// TIA Portal project "scl_6" (V18)

(* hardware
DEVICE "S7-1200 station_1"  S7-1200 Station
   slot 0: "Rack_0"  S7-1200 Rack  Rack  V1.0
   slot 1: "PLC_1"  CPU 1214C DC/DC/DC  6ES7 214-1AG40-0XB0  V4.6
*)

// ===== PLC "PLC_1"  CPU 1214C DC/DC/DC =====

VAR_GLOBAL   // PLC tag table "Default tag table"
   "START" AT %I0.0 : Bool;
   "STOP" AT %I0.1 : Bool;
   "MOTOR" AT %Q0.0 : Bool;
   "START1" AT %I0.2 : Bool;
   "START2" AT %I0.3 : Bool;
   "START3" AT %I0.4 : Bool;
   "SICAKLIK" AT %IW64 : Word;
   "BASINÇ" AT %IW66 : Word;
   "VALF1" AT %Q0.1 : Bool;
   "VALF2" AT %Q0.2 : Bool;
   "VALF3" AT %Q0.3 : Bool;
   "VALF4" AT %Q0.4 : Bool;
   "VALF5" AT %Q0.5 : Bool;
   "VALF6" AT %Q0.6 : Bool;
   "VALF7" AT %Q0.7 : Bool;
END_VAR

VAR_GLOBAL   // PLC tag table "Tag table_1"
   "ANALOG DEĞER" AT %IW68 : Int;
   "ANALOG DEĞER(1)" AT %IW70 : Int;
   "VALF 1" AT %Q1.0 : Bool;
   "VALF 2" AT %Q1.1 : Bool;
   "VALF 3" AT %Q1.2 : Bool;
   "VALF 4" AT %Q1.3 : Bool;
   "VALF 5" AT %Q1.4 : Bool;
   "VALF 6" AT %Q1.5 : Bool;
   "VALF 7" AT %Q1.6 : Bool;
   "DİGİTAL ÇIKIŞLAR" AT %QW0 : Word;
END_VAR

FUNCTION "Block_1" : Void   // FC1, SCL
{ S7_Optimized_Access := 'TRUE' }
VERSION : 0.1
BEGIN
   IF "START"=1 THEN
       // Statement section IF
       "MOTOR" := 1;
   ELSE
       // Statement section ELSE
       "MOTOR" := 0;
   END_IF;
END_FUNCTION

FUNCTION "Block_2" : Void   // FC2, SCL
{ S7_Optimized_Access := 'TRUE' }
VERSION : 0.1
BEGIN
   IF "START1"=1 THEN
       "VALF1":=1;
   ELSIF "START2"=1 THEN
       "VALF2":=1;
   ELSIF "START3"=1 THEN
       "VALF3" := 1;
   ELSE
       "VALF4":=1;

   END_IF;

   IF "SICAKLIK"<=23000 THEN
       "VALF5" := 1;

   ELSIF "SICAKLIK">=20000 THEN
       "VALF6":=1;
   ELSE
       "VALF7":=1;
   END_IF;
END_FUNCTION

FUNCTION "Block_3" : Void   // FC3, SCL
{ S7_Optimized_Access := 'TRUE' }
VERSION : 0.1
BEGIN
   "DİGİTAL ÇIKIŞLAR" := 0;
   CASE "ANALOG DEĞER(1)" OF
       5000..10000:  // Statement section case 1
           "VALF 1" := 1;
       10001..15000:  // Statement section case 2 to 4
           "VALF 2" := 1;
       15001..18000:
           "VALF 3" := 1;
       18001..22000:
           "VALF 4" := 1;

       ELSE  // Statement section ELSE
          "VALF 5":=1 ;
   END_CASE;
   CASE "ANALOG DEĞER" OF
       3000:  // Statement section case 1
           "VALF 6" := 1;
           "VALF 7" := 0;

       5000,10000,20000:  // Statement section case 2 to 4
           "VALF 6" := 0;
           "VALF 7" := 1;

   END_CASE;
END_FUNCTION

ORGANIZATION_BLOCK "Main"   // OB1, LAD, ProgramCycle
TITLE = "Main Program Sweep (Cycle)"
{ S7_Optimized_Access := 'TRUE' }
VERSION : 0.1
   VAR_INPUT
      Initial_Call : Bool;   // Initial call of this OB
      Remanence : Bool;   // =True, if remanent data are available
   END_VAR
BEGIN
END_ORGANIZATION_BLOCK